ABB RobotStudio station: ip_20230218-135010.rsstn

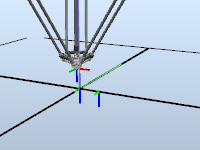
Station ip (saved by RobotStudio 7.0.8732.594)
Controller Controller1
  mechanical unit ROB_1: IRB360_1_800_4D_STD_03, 4 joints, base frame (0, 0, 0) mm, rotated rx 180 ry 0 rz 0 deg
Layout (positions relative to the parent item):
  - IRB360_1_800_4D_STD_03 [mechanism, from Robots\IRB360_1_800_4D_STD_03.rslib] at (0, 0, 0) mm, rotated rx 180 ry 0 rz 0 deg; joint values [0.6188, 0.5808, 0.0472, 0] (rad or m)
Targets, tools, work objects and paths stored in the station, written as RAPID:
! task T_ROB1
MODULE MainModule
  CONST robtarget ROBT_DEFAULT:=[[0,0,0],[0,1,0,0],[0,0,0,0],[9E+09,9E+09,9E+09,9E+09,9E+09,9E+09]];
  PROC main()
    MoveJ ROBT_DEFAULT,SD_DEFAULT,ZD_DEFAULT,tool0\WObj:=main_obj;
    MoveJ new_point,SD_DEFAULT,ZD_DEFAULT,tool0\WObj:=main_obj;
  ENDPROC
ENDMODULE

! task T_ROB1
MODULE CalibData
  TASK PERS wobjdata main_obj:=[FALSE,TRUE,"",[[0,0,-1150],[1,0,0,0]],[[0,0,0],[1,0,0,0]]];
ENDMODULE

! task T_ROB1
MODULE Module1
  CONST robtarget Target_10:=[[100,0,0],[0,1,0,0],[0,0,0,0],[9E+09,9E+09,9E+09,9E+09,9E+09,9E+09]];
ENDMODULE

